// TwinCAT 3 PLC project ScanRobot
// ProgramVersion: 3.1.4023.0
// libraries:
//   Tc2_Standard, * (Beckhoff Automation GmbH)
//   Tc2_System, * (Beckhoff Automation GmbH)
//   Tc2_Utilities, * (Beckhoff Automation GmbH)
//   Tc3_IotBase, * (Beckhoff Automation GmbH)
//   Tc3_Module, * (Beckhoff Automation GmbH)
// project tree:
//   DUTs/ MQTTSettings.TcDUT
//   / PlcTask.TcTTO (not stored)
//   POUs/ MAIN.TcPOU (not stored), MQTT.TcPOU

// ---- DUTs/MQTTSettings.TcDUT
TYPE MQTTSettings :
STRUCT
	//Broker info
	brokerIP : STRING := '78.27.125.143';
    brokerPort : UINT := 8885;
	brokerUsername : STRING := 'scanrobot';
	brokerPassword : STRING := 'kissa';
	
	//Client info
    clientId : STRING := 'plc';
	topicPub : STRING := 'beckhoff';
	topicSub : STRING := 'beckhoff';
	qos : TcIotMqttQos := TcIotMqttQos.AtMostOnceDelivery;	
	
	//TLS info
	caCertificateAbsolutePath : STRING := 'C:\Users\mikko\Desktop\folders\projects\scan_robot\twincat\certs\ca.crt';
	clientCertificateAbsolutePath : STRING := 'C:\Users\mikko\Desktop\folders\projects\scan_robot\twincat\certs\client.crt';
	clientKeyAbsolutePath : STRING := 'C:\Users\mikko\Desktop\folders\projects\scan_robot\twincat\certs\client.key';
END_STRUCT
END_TYPE

// ---- POUs/MQTT.TcPOU
FUNCTION_BLOCK MQTT
VAR_OUTPUT
	mqttClient : FB_IotMqttClient;
END_VAR
VAR
	mqttSettings : MQTTSettings;
END_VAR

METHOD PUBLIC configureMQTTClient
VAR_IN_OUT
END_VAR
mqttClient.sHostName := mqttSettings.brokerIP;
mqttClient.nHostPort := mqttSettings.brokerPort;
mqttClient.sClientId := mqttSettings.clientId;
mqttClient.sUserName := mqttSettings.brokerUsername;
mqttClient.sUserPassword := mqttSettings.brokerPassword;
mqttClient.stTLS.sCA := mqttSettings.caCertificateAbsolutePath;
mqttClient.stTLS.sCert := mqttSettings.clientCertificateAbsolutePath;
mqttClient.stTLS.sKeyFile := mqttSettings.clientKeyAbsolutePath;
END_METHOD

METHOD PUBLIC connect
mqttClient.Execute(bConnect := TRUE);
END_METHOD

METHOD PUBLIC isConnected : BOOL
isConnected := mqttClient.bConnected;
END_METHOD

METHOD PUBLIC publish : BOOL
VAR_INPUT
	msg : STRING;
END_VAR
mqttClient.Publish(sTopic:= mqttSettings.topicPub,
            pPayload:= ADR(msg),
            nPayloadSize:= LEN2(ADR(msg))+1,
            eQoS:= mqttSettings.qos,
            bRetain:= FALSE,
            bQueue:= FALSE
);
END_METHOD

METHOD PUBLIC publishWithTON
VAR_IN_OUT
	timer : TON;	
END_VAR
VAR_INPUT
	msg : STRING;
END_VAR
IF isConnected() THEN
    timer(IN:=TRUE);
    IF timer.Q THEN
        timer(IN:=FALSE);
     
        publish(msg := msg);
    END_IF
END_IF
END_METHOD

END_FUNCTION_BLOCK
